% RSLogix 500 project Project 8.RSS, saved by version 8.30.00.16 %
PROJECT "UNTITLED"    % processor: Bul.1763 MicroLogix 1100 Series B %

PROGRAM FILES
  LAD 2   15 rungs

DATA FILES
  O0 OUTPUT  4 elements
  I1 INPUT  6 elements
  S2 STATUS  66 elements
  B3 BINARY  1 elements
  T4 TIMER  1 elements
  C5 COUNTER  1 elements
  R6 CONTROL  1 elements
  N7 INTEGER  8 elements
  F8 FLOAT  3 elements

LADDER 2
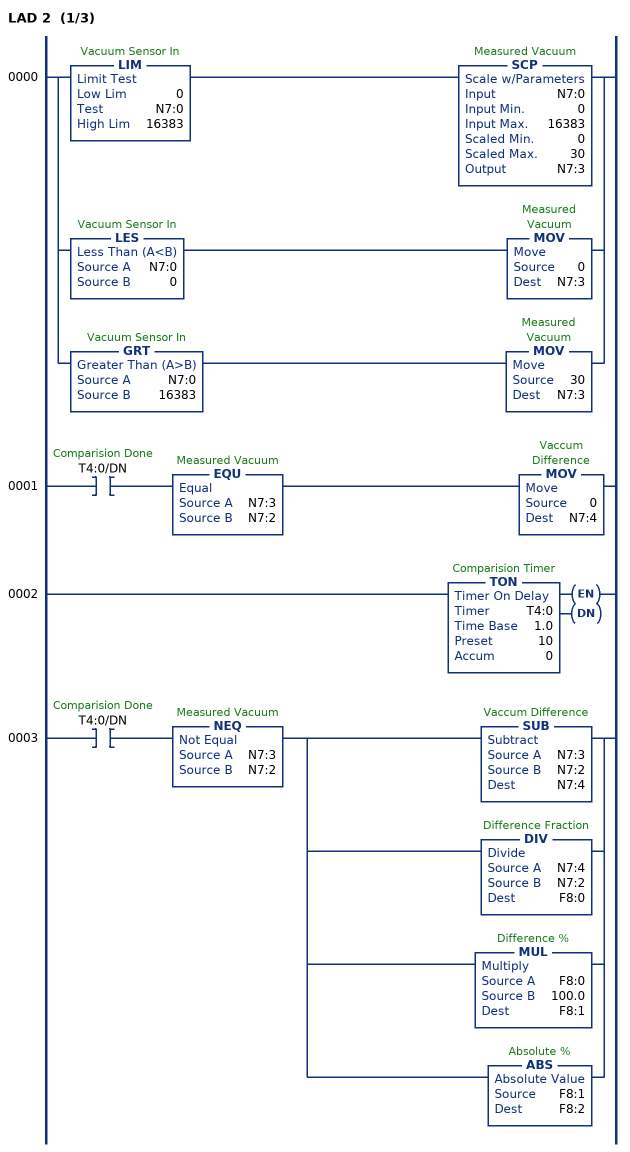
% Rung: 0 %
SOR BST LIM 0 N7:0 16383 SCP N7:0 0 16383 0 30 N7:3 NXB LES N7:0 0 MOV 0 N7:3 NXB GRT N7:0 16383 MOV 30 N7:3 BND EOR
%   N7:0  "Vacuum Sensor In" %
%   N7:3  "Measured Vacuum" %
% Rung: 1 %
SOR XIC T4:0/DN EQU N7:3 N7:2 MOV 0 N7:4 EOR
%   T4:0/DN  "Comparision Done" %
%   N7:3  "Measured Vacuum" %
%   N7:2  "Vacuum Setpoint" %
%   N7:4  "Vaccum Difference" %
% Rung: 2 %
SOR TON T4:0 1.0 10 0 EOR
%   T4:0  "Comparision Timer" %
% Rung: 3 %
SOR XIC T4:0/DN NEQ N7:3 N7:2 BST SUB N7:3 N7:2 N7:4 NXB DIV N7:4 N7:2 F8:0 NXB MUL F8:0 100.0 F8:1 NXB ABS F8:1 F8:2 BND EOR
%   T4:0/DN  "Comparision Done" %
%   N7:3  "Measured Vacuum" %
%   N7:2  "Vacuum Setpoint" %
%   N7:4  "Vaccum Difference" %
%   F8:0  "Difference Fraction" %
%   F8:1  "Difference %" %
%   F8:2  "Absolute %" %

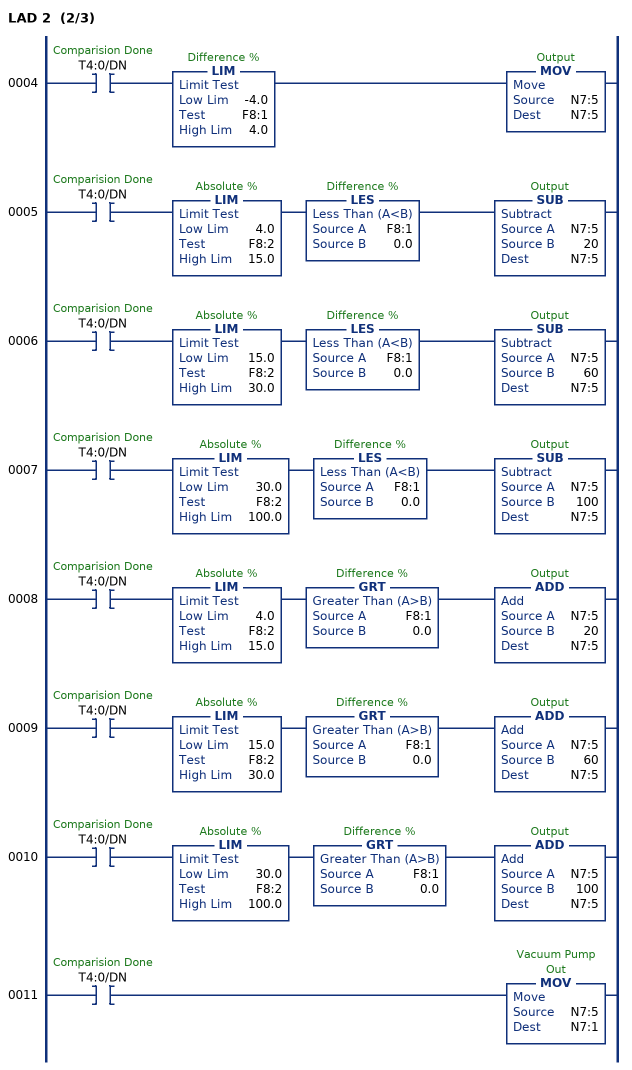
% Rung: 4 %
SOR XIC T4:0/DN LIM -4.0 F8:1 4.0 MOV N7:5 N7:5 EOR
%   T4:0/DN  "Comparision Done" %
%   F8:1  "Difference %" %
%   N7:5  "Output" %
% Rung: 5 %
SOR XIC T4:0/DN LIM 4.0 F8:2 15.0 LES F8:1 0.0 SUB N7:5 20 N7:5 EOR
%   T4:0/DN  "Comparision Done" %
%   F8:2  "Absolute %" %
%   F8:1  "Difference %" %
%   N7:5  "Output" %
% Rung: 6 %
SOR XIC T4:0/DN LIM 15.0 F8:2 30.0 LES F8:1 0.0 SUB N7:5 60 N7:5 EOR
%   T4:0/DN  "Comparision Done" %
%   F8:2  "Absolute %" %
%   F8:1  "Difference %" %
%   N7:5  "Output" %
% Rung: 7 %
SOR XIC T4:0/DN LIM 30.0 F8:2 100.0 LES F8:1 0.0 SUB N7:5 100 N7:5 EOR
%   T4:0/DN  "Comparision Done" %
%   F8:2  "Absolute %" %
%   F8:1  "Difference %" %
%   N7:5  "Output" %
% Rung: 8 %
SOR XIC T4:0/DN LIM 4.0 F8:2 15.0 GRT F8:1 0.0 ADD N7:5 20 N7:5 EOR
%   T4:0/DN  "Comparision Done" %
%   F8:2  "Absolute %" %
%   F8:1  "Difference %" %
%   N7:5  "Output" %
% Rung: 9 %
SOR XIC T4:0/DN LIM 15.0 F8:2 30.0 GRT F8:1 0.0 ADD N7:5 60 N7:5 EOR
%   T4:0/DN  "Comparision Done" %
%   F8:2  "Absolute %" %
%   F8:1  "Difference %" %
%   N7:5  "Output" %
% Rung: 10 %
SOR XIC T4:0/DN LIM 30.0 F8:2 100.0 GRT F8:1 0.0 ADD N7:5 100 N7:5 EOR
%   T4:0/DN  "Comparision Done" %
%   F8:2  "Absolute %" %
%   F8:1  "Difference %" %
%   N7:5  "Output" %
% Rung: 11 %
SOR XIC T4:0/DN MOV N7:5 N7:1 EOR
%   T4:0/DN  "Comparision Done" %
%   N7:5  "Output" %
%   N7:1  "Vacuum Pump Out" %

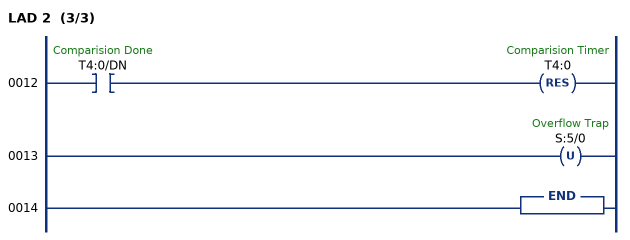
% Rung: 12 %
SOR XIC T4:0/DN RES T4:0 EOR
%   T4:0/DN  "Comparision Done" %
%   T4:0  "Comparision Timer" %
% Rung: 13 %
SOR OTU S:5/0 EOR
%   S:5/0  "Overflow Trap" %
% Rung: 14 %
SOR END EOR

OTHER DOCUMENTED ADDRESSES
  N7:6  "Difference %"
  N7:7  "Absolute %"

DATA TABLE (non-zero values as saved)
DATA T4
% .PRE .ACC %
% T4:0 % 10 0
DATA N7
% N7:0 % 0 0 15 0 0 0 0 0
